PROGRAM Homing
VAR
	horAxisHomingDone: BOOL := FALSE;
	rotAxisHomingDone: BOOL := FALSE;
	verAxisHomingDone: BOOL := FALSE;
END_VAR
VAR CONSTANT 
    HOME_SNAKE: INT := 1;
	HOME_SNAKEBOX: INT := 2;
	HOME_VERTICAL: INT := 3;
END_VAR

// State machine
CASE GVL.homingState OF
HOME_SNAKE:
	HAVL.axis.ReadStatus();
	
	IF horAxisHomingDone THEN
		HAVL.enable := FALSE;
		GVL.homingState := 2;
	ELSE
		HAVL.enable := TRUE;
	END_IF
	
	HAVL.axisPower(
		Axis:= HAVL.axis,
		Enable:= HAVL.enable,
		Enable_Positive:= HAVL.enable,
		Enable_Negative:= HAVL.enable,
		Override:= HAVL.override,
		BufferMode:= ,
		Options:= ,
		Status=> HAVL.running,
		Busy=> ,
		Active=> ,
		Error=> ,
		ErrorID=> HAVL.currentError
	);
	
	HAVL.axisHome(
		Axis:= HAVL.axis,
		Execute:= HAVL.execute,
		Position:= HAVL.homePosition,
		HomingMode:= MC_DefaultHoming,
		BufferMode:= ,
		Options:= ,
		bCalibrationCam:= HAVL.endStop,
		Done=> HAVL.done,
		Busy=> HAVL.busy,
		Active=> ,
		CommandAborted=> ,
		Error=> ,
		ErrorID=> HAVL.currentError
	);
	
	IF HAVL.running AND NOT(HAVL.busy) AND NOT(horAxisHomingDone) THEN
		HAVL.execute := TRUE;
	ELSE
		HAVL.execute := FALSE;
	END_IF
	
	IF HAVL.done THEN
		horAxisHomingDone := TRUE;
		RAVL.enable := TRUE;
	END_IF
		
HOME_SNAKEBOX:
	// do some invers motor shit	
	horAxisHomingDone := FALSE;
	
	RAVL.axis.ReadStatus();
	
	IF rotAxisHomingDone THEN
		RAVL.enable := FALSE;
		GVL.homingState := 3;
	ELSE
		RAVL.enable := TRUE;
	END_IF
	
	RAVL.axisPower(
		Axis:= RAVL.axis,
		Enable:= RAVL.enable,
		Enable_Positive:= RAVL.enable,
		Enable_Negative:= RAVL.enable,
		Override:= RAVL.override,
		BufferMode:= ,
		Options:= ,
		Status=> RAVL.running,
		Busy=> ,
		Active=> ,
		Error=> ,
		ErrorID=> RAVL.currentError
	);
	
	RAVL.axisHome(
		Axis:= RAVL.axis,
		Execute:= RAVL.execute,
		Position:= RAVL.homePosition,
		HomingMode:= MC_DefaultHoming,
		BufferMode:= ,
		Options:= ,
		bCalibrationCam:= RAVL.endStop,
		Done=> RAVL.done,
		Busy=> RAVL.busy,
		Active=> ,
		CommandAborted=> ,
		Error=> ,
		ErrorID=> RAVL.currentError
	);
	
	
	
	IF RAVL.running AND NOT(RAVL.busy) AND NOT(rotAxisHomingDone) THEN
		RAVL.execute := TRUE;
	ELSE
		RAVL.execute := FALSE;
	END_IF
	
	IF RAVL.done THEN
		rotAxisHomingDone := TRUE;
		//VAVL.enable := TRUE;
	END_IF
	
HOME_VERTICAL:
	//SAMELUR
	rotAxisHomingDone := FALSE;
	
	VAVL.axis.ReadStatus();
	
	IF verAxisHomingDone THEN
		VAVL.enable := FALSE;
		GVL.homingState := 1;
		GVL.stateGRAB := 0;
	ELSE
		VAVL.enable := TRUE;
	END_IF
	
	VAVL.axisPower(
		Axis:= VAVL.axis,
		Enable:= VAVL.enable,
		Enable_Positive:= VAVL.enable,
		Enable_Negative:= VAVL.enable,
		Override:= VAVL.override,
		BufferMode:= ,
		Options:= ,
		Status=> VAVL.running,
		Busy=> ,
		Active=> ,
		Error=> ,
		ErrorID=> VAVL.currentError
	);
	
	VAVL.axisHome(
		Axis:= VAVL.axis,
		Execute:= VAVL.execute,
		Position:= VAVL.homePosition,
		HomingMode:= MC_DefaultHoming,
		BufferMode:= ,
		Options:= ,
		bCalibrationCam:= NOT(VAVL.endStopBottom),
		Done=> VAVL.done,
		Busy=> VAVL.busy,
		Active=> ,
		CommandAborted=> ,
		Error=> ,
		ErrorID=> VAVL.currentError
	);
	
	IF VAVL.running AND NOT(VAVL.busy) AND NOT(verAxisHomingDone) THEN
		VAVL.execute := TRUE;
	ELSE
		VAVL.execute := FALSE;
	END_IF
	
	IF VAVL.done THEN
		verAxisHomingDone := TRUE;
	END_IF

ELSE
	// GRAB waiting for command
END_CASE

END_PROGRAM

(* stored: Version 1.1.0.1, ProductVersion 3.1.4024.6
   POU Homing: Id {8836339f-fb55-435b-a3e5-dd7a52c0a178}, SpecialFunc None *)
